PROGRAM HMI_System_Indicator
VAR
	bSystemFlag : BOOL;
END_VAR

IF
	GV_LIFT.ESTOP_INDICATOR_OUT AND GV_LIFT.ULTIMATE_LIMIT_INDICATOR_IN AND GV_LIFT.UP_LIMIT_INDICATOR_IN AND GV_LIFT.DOWN_LIMIT_INDICATOR_IN AND HMI.bSoftLimFlag AND HMI_Door_Toggle.bDoorFlag = FALSE AND HMI_Crush_Indicator.bCrushFlag = FALSE THEN
	bSystemFlag := TRUE;
ELSE
	bSystemFlag := FALSE;
END_IF

END_PROGRAM

(* stored: Version 1.1.0.1, ProductVersion 3.1.4022.12
   POU HMI_System_Indicator: Id {5deedf6c-fe35-4cf8-8e96-7ebcc8d7d603}, SpecialFunc None *)
